// TIA Portal V17 export
// export: Created 2023-02-26T22:28:46.7044738Z, ExportSetting WithDefaults, DisplayName Totally Integrated Automation Portal, DisplayVersion V17, DisplayName TIA Portal Openness, DisplayVersion V17, DisplayName TIA Portal Version Control Interface, DisplayVersion V17, DisplayName TIA Portal Test Suite Advanced, DisplayVersion V17, DisplayName STEP 7 Professional, DisplayVersion V17, DisplayName SIMATIC Energy Suite, DisplayVersion V17, DisplayName STEP 7 Safety, DisplayVersion V17, DisplayName WinCC Professional, DisplayVersion V17
DATA_BLOCK "ERR_EStop_DB"   // DB21
VERSION : 0.1
// stored: AutoNumber true, InstanceOfName ERR_EStop, InstanceOfType FB
"ERR_EStop"
   // VAR_INPUT
   //    EStopButton : Bool;
   //    ResetButton : Bool;
   // END_VAR
   // VAR_OUTPUT
   //    Error : Bool;
   // END_VAR
   // VAR
   //    P_ResetButton : Bool;
   // END_VAR
BEGIN
END_DATA_BLOCK
